// Mitsubishi GX Works2 project: LRI - PLC - AULA 12   PLC: Q03UDV

// task Task_01 (event TRUE, interval 0, priority 31): POU_01

PROGRAM POU_01
VAR
  Resultado : ARRAY [0..9] OF INT;
END_VAR
Resultado[0]:= st_Calculadora( TRUE , 40 , 5 , "+" );

Resultado[2]:= st_Calculadora_Case( TRUE , 40 , 5 , "*");

Resultado[3]:=st_Calculadora_Case( TRUE , 20 , 2 , "*" );
END_PROGRAM

FUNCTION st_Calculadora
VAR_INPUT
  x_Habilitar : BOOL;
  i_ValorUm : INT;
  i_ValorDois : INT;
  stg_Operador : STRING[32];
END_VAR

IF x_Habilitar THEN
		IF stg_Operador="+" THEN	
						st_Calculadora := i_ValorUm + i_ValorDois ;
						ELSIF stg_Operador="-" THEN
						st_Calculadora :=   i_ValorUm - i_ValorDois;
						ELSIF stg_Operador="*" THEN	
						st_Calculadora :=   i_ValorUm * i_ValorDois;
						ELSIF stg_Operador="/" THEN
						st_Calculadora :=  i_ValorUm / i_ValorDois ;
						ELSIF stg_Operador="M" OR stg_Operador="m" THEN
						st_Calculadora :=   i_ValorUm MOD i_ValorDois;
						ELSE
						st_Calculadora:= 32767;
					END_IF;
	END_IF;
END_FUNCTION

FUNCTION st_Calculadora_Case
VAR_INPUT
  x_Habilitar_Case : BOOL;
  i_ValorUm_Case : INT;
  i_ValorDois_Case : INT;
  stg_Operador_Case : STRING[32];
END_VAR
VAR
  i_Auxiliar_Case : INT;
END_VAR

IF x_Habilitar_Case THEN
	
		IF stg_Operador_Case="+" THEN	
						i_Auxiliar_Case:=0;
						
						ELSIF stg_Operador_Case="-" THEN
						i_Auxiliar_Case:=1;
						
						ELSIF stg_Operador_Case="*" THEN	
						i_Auxiliar_Case:=2;
						
						ELSIF stg_Operador_Case="/" THEN
						i_Auxiliar_Case:=3;
						
						ELSIF stg_Operador_Case="M" OR stg_Operador_Case="m" THEN
						i_Auxiliar_Case:=4;
						
						ELSE
						i_Auxiliar_Case:=5;
		END_IF;
		
		CASE i_Auxiliar_Case OF
		
		0:
			st_Calculadora_Case := i_ValorUm_Case + i_ValorDois_Case ;
		1:
		st_Calculadora_Case :=   i_ValorUm_Case - i_ValorDois_Case;
		2:
		st_Calculadora_Case :=   i_ValorUm_Case * i_ValorDois_Case;
		3:
			st_Calculadora_Case :=  i_ValorUm_Case / i_ValorDois_Case ;
		4:
		st_Calculadora_Case:=   i_ValorUm_Case MOD i_ValorDois_Case;
		5:
		st_Calculadora_Case:= 32767;
		END_CASE;	
		
END_IF;
END_FUNCTION
